(*
An identifier that uses reflection to generate a unique symbol path.
It simplifies the path by removing project, PLC, and tag segments.
Can be casted to `I_Arg` and `I_Component`.
Example:
- Reflection: proj.plc.MAIN.functionBlock[*]._tag
- Path: MAIN.functionBlock.5
*)
INTERFACE I_Tag EXTENDS I_Debug, I_RawComponent, I_Arg

// Read address path without Option segment.
PROPERTY Id : Str
GET
END_GET
END_PROPERTY

// Modify or read the optional segment.
PROPERTY Option : Str
GET
END_GET
END_PROPERTY

END_INTERFACE

(* stored: Version 1.1.0.1
   Itf I_Tag: Id {3b7d0464-054c-4855-8e00-e0918a18417d}
   Property Id: Id {a68c541f-7bc5-477f-8c26-6a17d7eb2271}
   Get Get: Id {8c83fc25-7b57-4b5d-9702-2e725bfd31a9}
   Property Option: Id {8c79c8bc-96ce-4254-84e1-a392e5aab50b}
   Get Get: Id {f7fa3efc-e0ec-4365-b02f-31a1cbfcb7b8} *)
